# EPICS StreamDevice protocol: Terminal/pot-switch.proto
terminator = CR LF;

info{
   out "ID?";
   in "%s";
}

getValue {
   out "POT?";
   in "%f";
}

getState{
   out "ROC?";
   in "%f:%s";
}
